(* IEC 61131-3 sources: altus-mobile/clpaltus/codigo, 3 files *)

(* ---- GVL_MODBUS.st ---- *)
(*
  ARQUIVO: GVL_MODBUS.st
  ONDE USAR: MasterTool > Application > UserGVLs > GVL_MODBUS
  O QUE FAZ: declara as variáveis usadas na comunicação Modbus RTU via RS-485

  IMPORTANTE: as variáveis MB_REG_KIT1 e MB_REG_KIT2 precisam ser mapeadas
  na configuração de hardware do MasterTool para os registradores do CLP escravo.
  Veja o GUIA_PASSO_A_PASSO.md seção "PARTE 3 — Configurar Modbus RS-485".
*)

VAR_GLOBAL

    (* ---------------------------------------------------------------
       Registradores enviados ao CLP escravo via Modbus RTU
       Cada WORD carrega 16 bits — usamos os 8 primeiros de cada um.

       MB_REG_KIT1 — bits mapeados para Kit 1:
         bit 0 = Q00 (pushbutton/1)    bit 4 = Q04 (switch/1)
         bit 1 = Q01 (pushbutton/2)    bit 5 = Q05 (switch/2)
         bit 2 = Q02 (pushbutton/3)    bit 6 = Q06 (switch/3)
         bit 3 = Q03 (pushbutton/4)    bit 7 = Q07 (switch/4)

       MB_REG_KIT2 — bits mapeados para Kit 2:
         bit 0 = Q08 (pushbutton/1)    bit 4 = Q12 (switch/1)
         bit 1 = Q09 (pushbutton/2)    bit 5 = Q13 (switch/2)
         bit 2 = Q10 (pushbutton/3)    bit 6 = Q14 (switch/3)
         bit 3 = Q11 (pushbutton/4)    bit 7 = Q15 (switch/4)
       --------------------------------------------------------------- *)
    MB_REG_KIT1 : WORD;   (* Registrador 40001 no CLP escravo *)
    MB_REG_KIT2 : WORD;   (* Registrador 40002 no CLP escravo *)

    (* Status da comunicação Modbus — para monitorar no MasterTool *)
    MB_CONNECTED : BOOL;  (* TRUE quando escravo responde *)
    MB_ERROR     : BOOL;  (* TRUE quando há falha de comunicação *)

END_VAR

(* ---- GVL_MQTT.st ---- *)
(*
  ARQUIVO: GVL_MQTT.st
  ONDE USAR: MasterTool > pasta MQTT > GVL_MQTT
  O QUE FAZ: declara todas as variáveis compartilhadas entre os programas MQTT
*)

VAR_GLOBAL

    (* Arrays internos da biblioteca LibMQTT — não mexa *)
    Pubs : ARRAY[1..gc_uiMaxPubs] OF MQTT_PUBLISH;
    Subs : ARRAY[1..gc_uiMaxSubs] OF MQTT_SUBSCRIBE;

    (* ---------------------------------------------------------------
       TÓPICOS — 16 no total (8 para Kit1, 8 para Kit2)
       A posição aqui define o índice usado nos outros programas.
       Publicar e assinar usam os MESMOS tópicos.
       --------------------------------------------------------------- *)
    MQTT_TOPICS : ARRAY[1..16] OF STRING := [
        (* Kit 1 - Botões (pushbutton) *)
        'altus/kit1/pushbutton/1',   (* pos 1  → Q00 / kit1Led1 *)
        'altus/kit1/pushbutton/2',   (* pos 2  → Q01 / kit1Led2 *)
        'altus/kit1/pushbutton/3',   (* pos 3  → Q02 / kit1Led3 *)
        'altus/kit1/pushbutton/4',   (* pos 4  → Q03 / kit1Led4 *)
        (* Kit 1 - Chaves (switch) *)
        'altus/kit1/switch/1',       (* pos 5  → Q04 / kit1Led5 *)
        'altus/kit1/switch/2',       (* pos 6  → Q05 / kit1Led6 *)
        'altus/kit1/switch/3',       (* pos 7  → Q06 / kit1Led7 *)
        'altus/kit1/switch/4',       (* pos 8  → Q07 / kit1Led8 *)
        (* Kit 2 - Botões (pushbutton) *)
        'altus/kit2/pushbutton/1',   (* pos 9  → Q08 / kit2Led1 *)
        'altus/kit2/pushbutton/2',   (* pos 10 → Q09 / kit2Led2 *)
        'altus/kit2/pushbutton/3',   (* pos 11 → Q10 / kit2Led3 *)
        'altus/kit2/pushbutton/4',   (* pos 12 → Q11 / kit2Led4 *)
        (* Kit 2 - Chaves (switch) *)
        'altus/kit2/switch/1',       (* pos 13 → Q12 / kit2Led5 *)
        'altus/kit2/switch/2',       (* pos 14 → Q13 / kit2Led6 *)
        'altus/kit2/switch/3',       (* pos 15 → Q14 / kit2Led7 *)
        'altus/kit2/switch/4'        (* pos 16 → Q15 / kit2Led8 *)
    ];

    (* Status internos — não mexa *)
    MQTT_FB_Pub_Status        : ARRAY[1..gc_uiMaxPubs] OF BOOL;
    MQTT_FB_Received_Messages : ARRAY[1..gc_uiMaxSubs] OF MQTT_RECEIVED;

    (* Payloads recebidos do app (o que chegou de cada tópico) *)
    SUBS_PAYLOADS : ARRAY[1..gc_uiMaxSubs] OF STRING;

    (* Payloads para publicar de volta (atualiza os LEDs do app) *)
    PUBS_PAYLOADS     : ARRAY[1..gc_uiMaxPubs] OF STRING;
    PUBS_PAYLOADS_OLD : ARRAY[1..gc_uiMaxPubs] OF STRING;

END_VAR

(* ---- MQTT.st ---- *)
(*
  ARQUIVO: MQTT.st
  ONDE USAR: MasterTool > pasta MQTT > MQTT (PRG)
  O QUE FAZ: configura a conexão com o broker Mosquitto e mantém ela ativa.

  !! ATENÇÃO !!
  Antes de carregar no CLP, você PRECISA trocar o IP abaixo.
  Para descobrir o IP do seu PC: abra o CMD e digite "ipconfig"
  Procure por "Endereço IPv4" (exemplo: 192.168.1.100)
*)

(* ===== SEÇÃO VAR — cole na parte de CIMA do editor ===== *)
(*
VAR
    MQTT_FB            : MQTT_CLIENT;
    MQTT_FB_Enable     : BOOL := TRUE;
    MQTT_FB_Error      : BOOL;
    MQTT_FB_State      : MQTT_STATES;
    MQTT_FB_Error_Code : MQTT_ERR_CODE;
    i                  : INT;
END_VAR
*)

(* ===== CÓDIGO — cole na parte de BAIXO do editor ===== *)

(* ------ TROQUE O IP AQUI ------
   sHostname = IP do PC onde o Mosquitto está rodando
   Exemplo:   '192.168.1.100'
   -------------------------------- *)
MQTT_FB_CONNECTION_CONFIG.sHostname     := '192.168.X.X';
MQTT_FB_CONNECTION_CONFIG.uiPort        := 1883;
MQTT_FB_CONNECTION_CONFIG.sClientId     := 'clp_xp340_kit1';
MQTT_FB_CONNECTION_CONFIG.bCleanSession := TRUE;

(* Aponta os arrays declarados na GVL_MQTT *)
MQTT_FB.PUBLISH   := Pubs;
MQTT_FB.SUBSCRIBE := Subs;

(* Habilita a função MQTT *)
MQTT_FB_Enable := MQTT_FB.Enable;

(* Lê os status de erro e conexão *)
MQTT_FB_Error             := MQTT_FB.ERROR;
MQTT_FB_State             := MQTT_FB.STATE;
MQTT_FB_Error_Code        := MQTT_FB.ERROR_CODE;
MQTT_FB_Pub_Status        := MQTT_FB.PUBLISH_STATUS;
MQTT_FB_Received_Messages := MQTT_FB.RECEIVED_MESSAGES;

(* Configura as assinaturas — o CLP vai escutar estes 8 tópicos *)
FOR i := 1 TO 8 DO
    Subs[i].eSubscribeTopic  := SUBSCRIBE_TOPICS[i];
    Subs[i].pbPayloadBuffer  := ADR(SUBS_PAYLOADS[i]);
    Subs[i].uiMaxPayloadSize := SIZEOF(SUBS_PAYLOADS[i]);
    Subs[i].eSubscribeQos    := MQTT_QOS_0;
END_FOR

(* Reconecta automaticamente se cair a conexão *)
IF MQTT_FB_Error THEN
    MQTT_FB_Enable := PULSE_55;
ELSE
    MQTT_FB_Enable := TRUE;
END_IF

(* Chama a função — deve ser a última linha *)
MQTT_FB();
